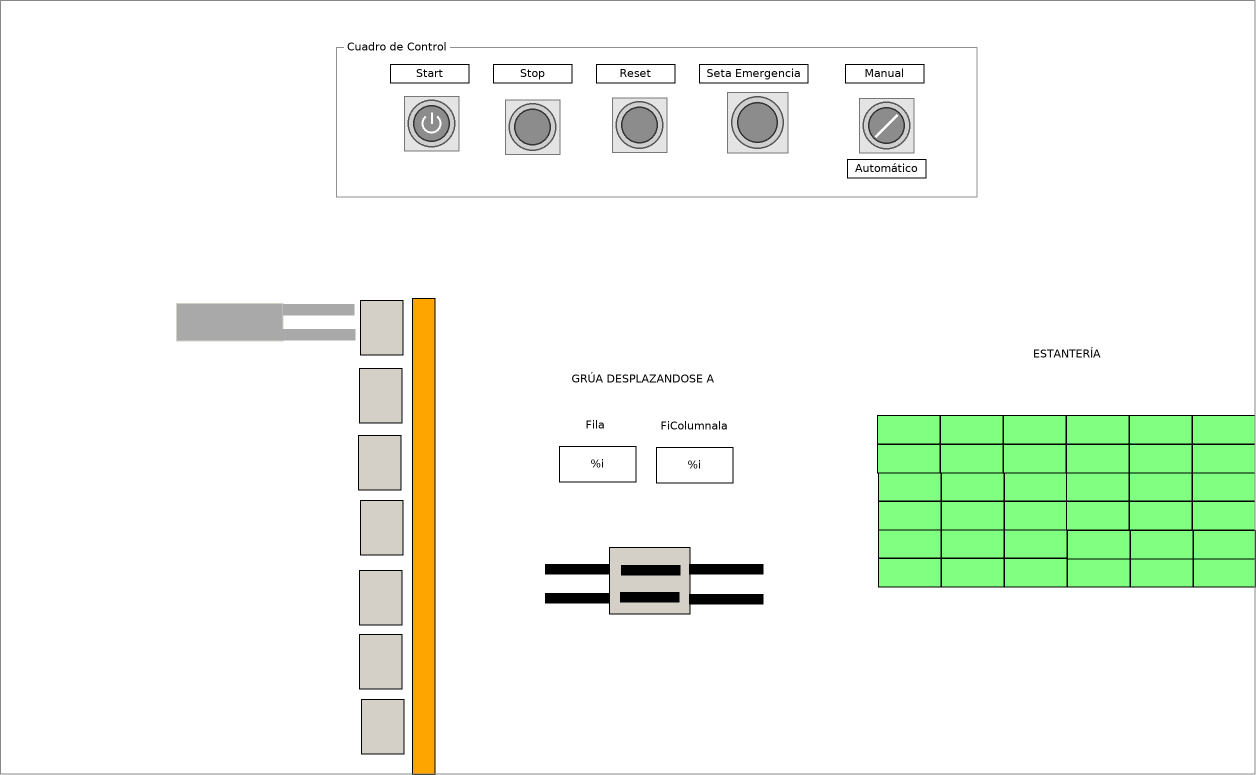
VISUALIZATION HMI  // 1256x775
    Rectangle (559,446 77x36), "%i", text variable: MAIN.filaEstanteria
    Label (580,410 30x30), "Fila"
    Rectangle (656,447 77x36), "%i", text variable: MAIN.colEstanteria
    Label (668,411 52x30), "FiColumnala"
    RoundedRectangle (878,558 63x29), colour toggle: GVLvar.baldasOcupadas[1,1], text list: 'equivalenciaBaldaOcupada', text index: GVLvar.baldasOcupadas[1][1]
        p2167032090: not GVLvar.baldasOcupadas[1][1]
        p3092690914: GVLvar.baldasOcupadas[1][1]
        toggle GVLvar.baldasOcupadas[1,1]
    Label (552,364 182x30), "GRÚA DESPLAZANDOSE A"
    Label (992,339 150x30), "ESTANTERÍA"
    GroupBox (336,39 641x158), "Cuadro de Control"
        PowerSwitch (64,57 63x55), variable: GVLvar.botonStart, behaviour: TOGGLE, style: Switch-PowerSwitch-Gray
        PushSwitch (169,58 55x60), variable: GVLvar.botonStop, behaviour: TOGGLE, style: Switch-PushSwitch-Gray
        PushSwitch (276,56 55x60), variable: GVLvar.botonReset, behaviour: TOGGLE, style: Switch-PushSwitch-Gray
        PushSwitchLed (390,53 63x61), variable: GVLvar.seta, behaviour: TOGGLE, style: Switch-PushSwitchLed-Gray
        Rectangle (54,25 79x19), "Start"
        Rectangle (157,25 79x19), "Stop"
        Rectangle (260,25 79x19), "Reset"
        Rectangle (363,25 109x19), "Seta Emergencia"
        Rectangle (509,25 79x19), "Manual"
        Rectangle (511,120 79x19), "Automático"
        RotarySwitch (523,59 55x55), variable: GVLvar.modoManual, behaviour: TOGGLE, style: Switch-RotarySwitch-Gray
    Rectangle (176,303 107x38), colour toggle: GVLvar.cinta
        toggle GVLvar.cinta
    Rectangle (283,304 71x11), colour toggle: GVLvar.cintaTransportadoraPalet
        toggle GVLvar.cintaTransportadoraPalet
    Rectangle (282,329 73x11), colour toggle: GVLvar.cintaTransportadoraPalet
        toggle GVLvar.cintaTransportadoraPalet
    Rectangle (412,298 23x477)
    Rectangle (609,547 81x67)
    Rectangle (545,593 64x10), colour toggle: GVLvar.moveForksRight, invisible if: Not GVLvar.moveForksRight
        toggle GVLvar.moveForksRight
    Rectangle (689,594 74x10), colour toggle: GVLvar.moveForksLeft, invisible if: Not GVLvar.moveForksLeft
        toggle GVLvar.moveForksLeft
    RoundedRectangle (941,558 63x29), colour toggle: GVLvar.baldasOcupadas[1,2], text list: 'equivalenciaBaldaOcupada', text index: GVLvar.baldasOcupadas[1][1]
        p2167032090: not GVLvar.baldasOcupadas[1][1]
        p3092690914: GVLvar.baldasOcupadas[1][1]
        toggle GVLvar.baldasOcupadas[1,2]
    RoundedRectangle (1004,558 63x29), colour toggle: GVLvar.baldasOcupadas[1,3], text list: 'equivalenciaBaldaOcupada', text index: GVLvar.baldasOcupadas[1][1]
        p2167032090: not GVLvar.baldasOcupadas[1][1]
        p3092690914: GVLvar.baldasOcupadas[1][1]
        toggle GVLvar.baldasOcupadas[1,3]
    RoundedRectangle (878,529 63x29), colour toggle: GVLvar.baldasOcupadas[2,1], text list: 'equivalenciaBaldaOcupada', text index: GVLvar.baldasOcupadas[1][1]
        p2167032090: not GVLvar.baldasOcupadas[1][1]
        p3092690914: GVLvar.baldasOcupadas[1][1]
        toggle GVLvar.baldasOcupadas[2,1]
    RoundedRectangle (941,529 63x29), colour toggle: GVLvar.baldasOcupadas[2,2], text list: 'equivalenciaBaldaOcupada', text index: GVLvar.baldasOcupadas[1][1]
        p2167032090: not GVLvar.baldasOcupadas[1][1]
        p3092690914: GVLvar.baldasOcupadas[1][1]
        toggle GVLvar.baldasOcupadas[2,2]
    RoundedRectangle (1004,529 63x29), colour toggle: GVLvar.baldasOcupadas[2,3], text list: 'equivalenciaBaldaOcupada', text index: GVLvar.baldasOcupadas[1][1]
        p2167032090: not GVLvar.baldasOcupadas[1][1]
        p3092690914: GVLvar.baldasOcupadas[1][1]
        toggle GVLvar.baldasOcupadas[2,3]
    RoundedRectangle (878,501 63x29), colour toggle: GVLvar.baldasOcupadas[3,1], text list: 'equivalenciaBaldaOcupada', text index: GVLvar.baldasOcupadas[1][1]
        p2167032090: not GVLvar.baldasOcupadas[1][1]
        p3092690914: GVLvar.baldasOcupadas[1][1]
        toggle GVLvar.baldasOcupadas[3,1]
    RoundedRectangle (941,501 63x29), colour toggle: GVLvar.baldasOcupadas[3,2], text list: 'equivalenciaBaldaOcupada', text index: GVLvar.baldasOcupadas[1][1]
        p2167032090: not GVLvar.baldasOcupadas[1][1]
        p3092690914: GVLvar.baldasOcupadas[1][1]
        toggle GVLvar.baldasOcupadas[3,2]
    RoundedRectangle (1004,501 63x29), colour toggle: GVLvar.baldasOcupadas[3,3], text list: 'equivalenciaBaldaOcupada', text index: GVLvar.baldasOcupadas[1][1]
        p2167032090: not GVLvar.baldasOcupadas[1][1]
        p3092690914: GVLvar.baldasOcupadas[1][1]
        toggle GVLvar.baldasOcupadas[3,3]
    RoundedRectangle (878,472 63x29), colour toggle: GVLvar.baldasOcupadas[4,1], text list: 'equivalenciaBaldaOcupada', text index: GVLvar.baldasOcupadas[1][1]
        p2167032090: not GVLvar.baldasOcupadas[1][1]
        p3092690914: GVLvar.baldasOcupadas[1][1]
        toggle GVLvar.baldasOcupadas[1,1]
    RoundedRectangle (941,472 63x29), colour toggle: GVLvar.baldasOcupadas[4,2], text list: 'equivalenciaBaldaOcupada', text index: GVLvar.baldasOcupadas[1][1]
        p2167032090: not GVLvar.baldasOcupadas[1][1]
        p3092690914: GVLvar.baldasOcupadas[1][1]
        toggle GVLvar.baldasOcupadas[1,2]
    RoundedRectangle (1004,472 63x29), colour toggle: GVLvar.baldasOcupadas[4,3], text list: 'equivalenciaBaldaOcupada', text index: GVLvar.baldasOcupadas[1][1]
        p2167032090: not GVLvar.baldasOcupadas[1][1]
        p3092690914: GVLvar.baldasOcupadas[1][1]
        toggle GVLvar.baldasOcupadas[4,3]
    RoundedRectangle (877,444 63x29), colour toggle: GVLvar.baldasOcupadas[5,1], text list: 'equivalenciaBaldaOcupada', text index: GVLvar.baldasOcupadas[1][1]
        p2167032090: not GVLvar.baldasOcupadas[1][1]
        p3092690914: GVLvar.baldasOcupadas[1][1]
        toggle GVLvar.baldasOcupadas[5,1]
    RoundedRectangle (940,444 63x29), colour toggle: GVLvar.baldasOcupadas[5,2], text list: 'equivalenciaBaldaOcupada', text index: GVLvar.baldasOcupadas[1][1]
        p2167032090: not GVLvar.baldasOcupadas[1][1]
        p3092690914: GVLvar.baldasOcupadas[1][1]
        toggle GVLvar.baldasOcupadas[5,2] p2164770859=TRUE
    RoundedRectangle (1003,444 63x29), colour toggle: GVLvar.baldasOcupadas[5,3], text list: 'equivalenciaBaldaOcupada', text index: GVLvar.baldasOcupadas[1][1]
        p2167032090: not GVLvar.baldasOcupadas[1][1]
        p3092690914: GVLvar.baldasOcupadas[1][1]
        toggle GVLvar.baldasOcupadas[5,3]
    RoundedRectangle (877,415 63x29), colour toggle: GVLvar.baldasOcupadas[6,1], text list: 'equivalenciaBaldaOcupada', text index: GVLvar.baldasOcupadas[1][1]
        p2167032090: not GVLvar.baldasOcupadas[1][1]
        p3092690914: GVLvar.baldasOcupadas[1][1]
        toggle GVLvar.baldasOcupadas[6,1]
    RoundedRectangle (940,415 63x29), colour toggle: GVLvar.baldasOcupadas[6,2], text list: 'equivalenciaBaldaOcupada', text index: GVLvar.baldasOcupadas[1][1]
        p2167032090: not GVLvar.baldasOcupadas[1][1]
        p3092690914: GVLvar.baldasOcupadas[1][1]
        toggle GVLvar.baldasOcupadas[6,2]
    RoundedRectangle (1003,415 63x29), colour toggle: GVLvar.baldasOcupadas[6,3], text list: 'equivalenciaBaldaOcupada', text index: GVLvar.baldasOcupadas[1][1]
        p2167032090: not GVLvar.baldasOcupadas[1][1]
        p3092690914: GVLvar.baldasOcupadas[1][1]
        toggle GVLvar.baldasOcupadas[6,3]
    Rectangle (545,564 64x10), colour toggle: GVLvar.moveForksRight, invisible if: Not GVLvar.moveForksRight
        toggle GVLvar.moveForksRight
    Rectangle (689,564 74x10), colour toggle: GVLvar.moveForksLeft, invisible if: Not GVLvar.moveForksLeft
        toggle GVLvar.moveForksLeft
    Rectangle (360,300 43x55), invisible if: Not MAIN.reposo
    Rectangle (359,368 43x55), invisible if: Not (MAIN.colEstanteria =1)
    Rectangle (358,435 43x55), invisible if: Not (MAIN.colEstanteria = 2)
    Rectangle (360,500 43x55), invisible if: Not (MAIN.colEstanteria =3)
    Rectangle (359,570 43x55), invisible if: Not (MAIN.colEstanteria =4)
    Rectangle (359,634 43x55), invisible if: Not (MAIN.colEstanteria =5)
    Rectangle (361,699 43x55), invisible if: Not (MAIN.colEstanteria =6)
    Rectangle (620,592 59x10), colour toggle: GVLvar.moveForksRight, invisible if: Not GVLvar.forkMiddleLimit
        toggle GVLvar.moveForksRight
    RoundedRectangle (1067,558 63x29), text list: 'equivalenciaBaldaOcupada', text index: GVLvar.baldasOcupadas[1][1]
        p2167032090: not GVLvar.baldasOcupadas[1][1]
        p3092690914: GVLvar.baldasOcupadas[1][1]
    RoundedRectangle (1067,530 63x29), text list: 'equivalenciaBaldaOcupada', text index: GVLvar.baldasOcupadas[1][1]
        p2167032090: not GVLvar.baldasOcupadas[1][1]
        p3092690914: GVLvar.baldasOcupadas[1][1]
    RoundedRectangle (1066,501 63x29), text list: 'equivalenciaBaldaOcupada', text index: GVLvar.baldasOcupadas[1][1]
        p2167032090: not GVLvar.baldasOcupadas[1][1]
        p3092690914: GVLvar.baldasOcupadas[1][1]
    RoundedRectangle (1066,472 63x29), text list: 'equivalenciaBaldaOcupada', text index: GVLvar.baldasOcupadas[1][1]
        p2167032090: not GVLvar.baldasOcupadas[1][1]
        p3092690914: GVLvar.baldasOcupadas[1][1]
    RoundedRectangle (1066,444 63x29), text list: 'equivalenciaBaldaOcupada', text index: GVLvar.baldasOcupadas[1][1]
        p2167032090: not GVLvar.baldasOcupadas[1][1]
        p3092690914: GVLvar.baldasOcupadas[1][1]
    RoundedRectangle (1066,415 63x29), text list: 'equivalenciaBaldaOcupada', text index: GVLvar.baldasOcupadas[1][1]
        p2167032090: not GVLvar.baldasOcupadas[1][1]
        p3092690914: GVLvar.baldasOcupadas[1][1]
    RoundedRectangle (1130,558 63x29), text list: 'equivalenciaBaldaOcupada', text index: GVLvar.baldasOcupadas[1][1]
        p2167032090: not GVLvar.baldasOcupadas[1][1]
        p3092690914: GVLvar.baldasOcupadas[1][1]
    RoundedRectangle (1130,530 63x29), text list: 'equivalenciaBaldaOcupada', text index: GVLvar.baldasOcupadas[1][1]
        p2167032090: not GVLvar.baldasOcupadas[1][1]
        p3092690914: GVLvar.baldasOcupadas[1][1]
    RoundedRectangle (1129,501 63x29), text list: 'equivalenciaBaldaOcupada', text index: GVLvar.baldasOcupadas[1][1]
        p2167032090: not GVLvar.baldasOcupadas[1][1]
        p3092690914: GVLvar.baldasOcupadas[1][1]
    RoundedRectangle (1129,472 63x29), text list: 'equivalenciaBaldaOcupada', text index: GVLvar.baldasOcupadas[1][1]
        p2167032090: not GVLvar.baldasOcupadas[1][1]
        p3092690914: GVLvar.baldasOcupadas[1][1]
    RoundedRectangle (1129,444 63x29), text list: 'equivalenciaBaldaOcupada', text index: GVLvar.baldasOcupadas[1][1]
        p2167032090: not GVLvar.baldasOcupadas[1][1]
        p3092690914: GVLvar.baldasOcupadas[1][1]
    RoundedRectangle (1129,415 63x29), text list: 'equivalenciaBaldaOcupada', text index: GVLvar.baldasOcupadas[1][1]
        p2167032090: not GVLvar.baldasOcupadas[1][1]
        p3092690914: GVLvar.baldasOcupadas[1][1]
    RoundedRectangle (1193,558 63x29), text list: 'equivalenciaBaldaOcupada', text index: GVLvar.baldasOcupadas[1][1]
        p2167032090: not GVLvar.baldasOcupadas[1][1]
        p3092690914: GVLvar.baldasOcupadas[1][1]
    RoundedRectangle (1193,530 63x29), text list: 'equivalenciaBaldaOcupada', text index: GVLvar.baldasOcupadas[1][1]
        p2167032090: not GVLvar.baldasOcupadas[1][1]
        p3092690914: GVLvar.baldasOcupadas[1][1]
    RoundedRectangle (1192,501 63x29), text list: 'equivalenciaBaldaOcupada', text index: GVLvar.baldasOcupadas[1][1]
        p2167032090: not GVLvar.baldasOcupadas[1][1]
        p3092690914: GVLvar.baldasOcupadas[1][1]
    RoundedRectangle (1192,472 63x29), text list: 'equivalenciaBaldaOcupada', text index: GVLvar.baldasOcupadas[1][1]
        p2167032090: not GVLvar.baldasOcupadas[1][1]
        p3092690914: GVLvar.baldasOcupadas[1][1]
    RoundedRectangle (1192,444 63x29), text list: 'equivalenciaBaldaOcupada', text index: GVLvar.baldasOcupadas[1][1]
        p2167032090: not GVLvar.baldasOcupadas[1][1]
        p3092690914: GVLvar.baldasOcupadas[1][1]
    RoundedRectangle (1192,415 63x29), text list: 'equivalenciaBaldaOcupada', text index: GVLvar.baldasOcupadas[1][1]
        p2167032090: not GVLvar.baldasOcupadas[1][1]
        p3092690914: GVLvar.baldasOcupadas[1][1]
    Rectangle (621,565 59x10), colour toggle: GVLvar.moveForksRight, invisible if: Not GVLvar.forkMiddleLimit
        toggle GVLvar.moveForksRight
END_VISUALIZATION

(* stored: Version 1.1.0.1, ProductVersion 3.1.4024.15
   Visu HMI: Id {bfaba427-f570-4759-8e68-a2391132dc32} *)
